// TIA Portal V19 export
TYPE "LAF_typeXXXMaintanceParameters"
// stored: Access Published
   STRUCT
      upperVel : LReal;   // 维护速度上限
      vel : LReal;   // 维护速度设定值，画面做限制根据上限值如果超了不允许输入
      acc : LReal;
      dec : LReal;
   END_STRUCT;
END_TYPE
